FUNCTION_BLOCK E_SELECT_4 (* selection between two events based on boolean input G (4 channels, generic FB) *)
  (* Standard: 61499-1 Annex A; Classification: event function block; Function: Selection of events (4 channels); Description: Copyright (c) 2017, 2026 fortiss GmbH, HR Agrartechnik GmbH This program and the accompanying materials are made available under the terms of the Eclipse Public License 2.0 which is available at https://www.eclipse.org/legal/epl-2.0/ SPDX-License-Identifier: EPL-2.0 Some portions generated by Gemini CLI *)
  (* Version 1.0, 2026-02-01, Franz Höpfinger, HR Agrartechnik GmbH, Initial creation based on E_SELECT and E_SPLIT_3 *)
  PACKAGE iec61499::events;
  {SET_ATTRIBUTE(eclipse4diac::core::GenericClassName, 'GEN_E_SELECT')}
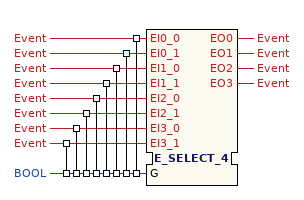
  EVENT_INPUT
    EI0_0 WITH G; (* Channel 0: Input event, selected when G=0 *)
    EI0_1 WITH G; (* Channel 0: Input event, selected when G=1 *)
    EI1_0 WITH G; (* Channel 1: Input event, selected when G=0 *)
    EI1_1 WITH G; (* Channel 1: Input event, selected when G=1 *)
    EI2_0 WITH G; (* Channel 2: Input event, selected when G=0 *)
    EI2_1 WITH G; (* Channel 2: Input event, selected when G=1 *)
    EI3_0 WITH G; (* Channel 3: Input event, selected when G=0 *)
    EI3_1 WITH G; (* Channel 3: Input event, selected when G=1 *)
  END_EVENT
  EVENT_OUTPUT
    EO0; (* Channel 0: Output Event *)
    EO1; (* Channel 1: Output Event *)
    EO2; (* Channel 2: Output Event *)
    EO3; (* Channel 3: Output Event *)
  END_EVENT
  VAR_INPUT
    G : BOOL; (* Select EIn_0 when G=0, EIn_1 when G=1 *)
  END_VAR
END_FUNCTION_BLOCK
